(* This FB is use to controll two axis to gear in move at the same time 
*)
FUNCTION_BLOCK FB_XY_Move EXTENDS FB_ActionBasic
VAR_INPUT
	xExecute : BOOL;
	xAbort : BOOL;
	xReset :BOOL;
	AxisX_No : AxisNo;
	AxisY_No : AxisNo;
	
    TimeOut     : LREAL := 30; // Unit : s
END_VAR
VAR_OUTPUT
	xAborted : BOOL;
END_VAR
VAR
	StateBehavior : CBML.ETrigATo;
	CurrentPosData :ST_PositionTable;
	uiCyclicStep :UINT;
END_VAR

THIS^.IBehaviourModel := StateBehavior;
StateBehavior(xExecute := xExecute,
              xAbort := xAbort,
              udiTimeOut := LREAL_TO_UDINT(TimeOut * 1000000),
              xDone => xDone,
              xBusy => xBusy,
              xError => xError,
              xAborted => xAborted);

METHOD CleanupAction
VAR_INPUT
    xAbortProposed : BOOL;
    iErrorIDProposed: INT;
END_VAR
VAR_OUTPUT
    xComplete : BOOL := TRUE;
    xAbort: BOOL := xAbortProposed;
 	iErrorID : INT := iErrorIDProposed;
END_VAR
END_METHOD

METHOD CyclicAction
VAR_INPUT
    itfTimingController : CBML.ITimingController;
END_VAR
VAR_OUTPUT
    xComplete : BOOL := TRUE;
    iErrorID : INT := 0;
END_VAR
xComplete := FALSE;
END_METHOD

METHOD ExitAction
VAR_INPUT
    xAfterCleanup : BOOL;
    xInCopyCode : BOOL;
END_VAR
END_METHOD

METHOD ResetAction
VAR_OUTPUT
    xComplete : BOOL := TRUE;
END_VAR
END_METHOD

METHOD StartAction
VAR_OUTPUT
    xComplete : BOOL := TRUE;
	iErrorID : INT := 0;
END_VAR

VAR_INST
	AxisX_Ready :BOOL;
	AxisY_Ready :BOOL;
END_VAR
xComplete := FALSE;
uiCyclicStep := 0;
AxisX_Ready := FUN_CheckAxisAllowMove(AxisNo := AxisX_No);
AxisY_Ready := FUN_CheckAxisAllowMove(AxisNo := AxisY_No);

IF NOT AxisX_Ready THEN
	iErrorID := 2; // AxisX not ready
ELSIF NOT AxisY_Ready THEN
	iErrorID := 3; // AxisY not Ready
ELSIF AxisX_Ready AND AxisY_Ready THEN
	iErrorID := 0;
	xComplete := TRUE;
END_IF
END_METHOD

END_FUNCTION_BLOCK

(* stored: Version 1.1.0.1, ProductVersion 3.1.4024.13
   POU FB_XY_Move: Id {7f40aa0d-a28d-4517-b739-f2e8fa92d1be}, SpecialFunc None
   Method CleanupAction: Id {3a621df1-113b-4f9e-a14e-8a04cdebf6ff}
   Method CyclicAction: Id {fe2941f7-08ab-4342-8b8b-3eec14f90537}
   Method ExitAction: Id {7b4b060a-fb2a-4653-868a-c80b8753cd1c}
   Method ResetAction: Id {edc5b0e2-99a0-4749-a94f-c1fd6583cde1}
   Method StartAction: Id {3e150b83-5177-4109-9189-ed341698d106} *)
